RoboDK station: Prep Stacji Filip.rdk

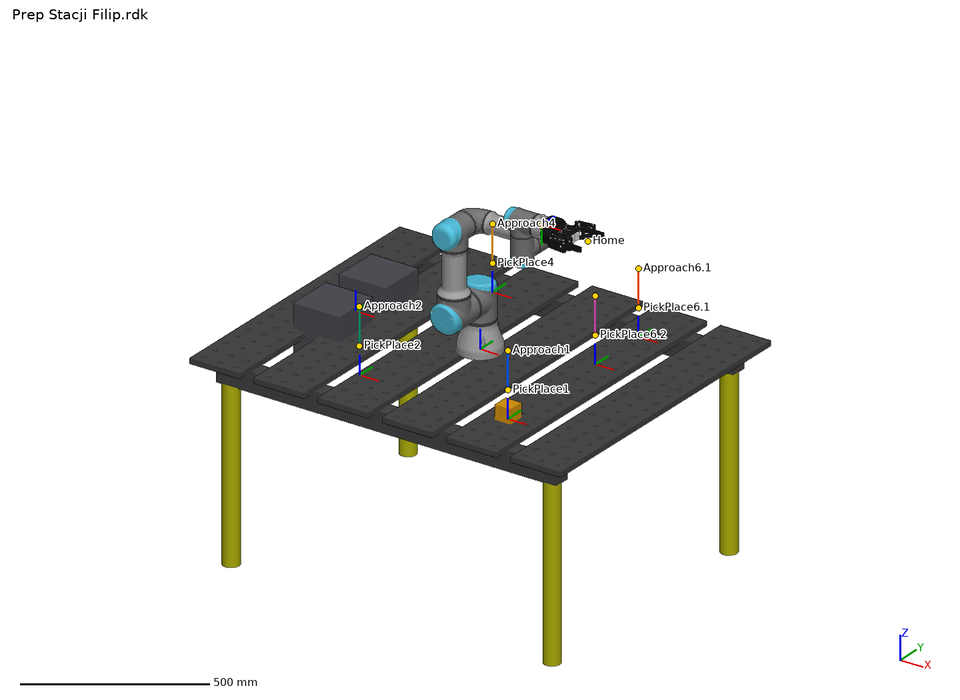
[picture v0: the station drawn from its stored meshes, robots at their saved joint values, targets as dots, program paths as lines]
Station Prep Stacji Filip. Poses are relative to the parent item; angles as X-Y-Z fixed-axis rotations.
  - frame UR3 Base at (0, 0, 0) mm
    - robot UR3: 6 axes, payload 3 kg, reach 500 mm, repeatability 0.1 mm, weight 11 kg
        modified DH rows (alpha deg, a mm, theta deg, d mm): 0, 0, 0, 151.9; 90, 0, 180, 0; 0, 243.65, 0, 0; 0, 213, 0, 110.4; -90, 0, 0, 83.4; 90, 0, 180, 82.4
        joint limits [-360, -360, -360, -360, -360, -360] to [360, 360, 360, 360, 360, 360]; home [0, -90, -90, 0, 90, 0]; saved at [0, -90, -90, 0, 90, 0]
      - tool Gripper, TCP at (0, 0, 130) mm, size 147.4 x 146.8 x 75 mm
    - object Table at (0, 0, 0) mm, size 1193.8 x 965.2 x 609.6 mm, geometry from welding_table.sld
    - target Home (Cartesian target) at (425.4, -110.4, 478.95) mm, rotated rx -90 ry 0 rz -90 deg; joints [0, -90, -90, 0, 90, 0] of UR3
    - object Vise_1 at (-400, 105, 0) mm, size 150 x 150 x 150 mm, geometry from box.sld
    - object Vise_2 at (-400, -105, 0) mm, size 150 x 150 x 150 mm, geometry from box.sld
  - frame Grab_Blank at (300, -300, 0) mm
    - target Approach1 (Cartesian target) at (0, 0, 200) mm, rotated rx 179.78 ry -0.22 rz -90 deg; joints [-29.763, -119.152, -47.872, -103.057, 89.704, -29.763] of UR3
    - target PickPlace1 (Cartesian target) at (0, 0, 85) mm, rotated rx 179.78 ry -0.22 rz -90 deg; joints [120.071, -59.59, 77.288, -107.776, -90.297, -59.929] of UR3
  - frame Blank_Buffer at (-170, -310, 0) mm
    - target Approach2 (Cartesian target) at (0, 0, 200) mm, rotated rx 179.78 ry -0.22 rz 90 deg; joints [-119.875, -118.751, -48.653, -102.3, 89.919, -119.875] of UR3
    - target PickPlace2 (Cartesian target) at (0, 0, 85) mm, rotated rx 179.78 ry -0.22 rz 90 deg; joints [-119.875, -120.162, -77.775, -71.767, 89.919, -119.875] of UR3
  - frame Workpiece_Holder at (-400, 0, 0) mm
  - frame Workpiece_Buffer at (-170, 300, 0) mm
    - target Approach4 (Cartesian target) at (0, 0, 200) mm, rotated rx 179.78 ry -0.22 rz 90 deg; joints [-209.763, -119.154, -47.869, -103.059, 89.704, -29.763] of UR3
    - target PickPlace4 (Cartesian target) at (0, 0, 85) mm, rotated rx 179.78 ry -0.22 rz 90 deg; joints [-209.763, -120.393, -77.248, -72.441, 89.704, -29.763] of UR3
  - frame Inspection_Point at (-47.33, 351.68, 211.92) mm, rotated rx -90 ry 0 rz 0 deg
    - target Inspekcja (Cartesian target) at (4.05, 0, -6.89) mm, rotated rx 0 ry 1.16 rz 0 deg; joints [161.436, -62.355, -137.519, -160.126, -17.407, 180] of UR3
    - target Inspekcja2 (Cartesian target) at (4.12, -0.12, -6.97) mm, rotated rx -0.02 ry -1.17 rz -180 deg; joints [161.482, -62.272, -137.542, -160.119, -17.348, -0.064] of UR3
    - target Inspekcja3 (Cartesian target) at (4.12, -0.12, -6.97) mm, rotated rx 0.02 ry 1.17 rz 0.01 deg; joints [161.482, -62.272, -137.542, -160.119, -17.348, 179.946] of UR3
  - frame Reject_Workpiece at (300, 300, 0) mm
    - target Approach6.1 (Cartesian target) at (0, 0, 200) mm, rotated rx 179.78 ry -0.22 rz -90 deg; joints [60.042, -119.541, -47.172, -103.583, 90.08, 60.041] of UR3
    - target PickPlace6.1 (Cartesian target) at (0, 0, 85) mm, rotated rx 179.78 ry -0.22 rz -90 deg; joints [60.042, -120.641, -76.761, -72.895, 90.08, 60.041] of UR3
  - frame Approve_Workpiece at (300, 100, 0) mm
    - target Approach6.2 (Cartesian target) at (0, 0, 200) mm, rotated rx 179.78 ry -0.22 rz -90 deg; joints [38.892, -90.405, -84.937, -94.964, 89.967, 38.892] of UR3
    - target PickPlace6.2 (Cartesian target) at (0, 0, 85) mm, rotated rx 179.78 ry -0.22 rz -90 deg; joints [38.892, -95.685, -111.257, -63.363, 89.967, 38.892] of UR3
  - program ResetStation (1 instructions, listed below)
  - program Pick1 (6 instructions, listed below)
  - program Pick2 (6 instructions, listed below)
  - program Place2 (6 instructions, listed below)
  - program Pick4 (6 instructions, listed below)
  - program Place4 (6 instructions, listed below)
  - program Inspekcja (5 instructions, listed below)
  - program Pick6.1 (6 instructions, listed below)
  - program Place6.1 (6 instructions, listed below)
  - program Pick6.2 (6 instructions, listed below)
  - program Place6.2 (6 instructions, listed below)
  - program main (8 instructions, listed below)
  - object Workpiece_50mm at (300, -300, 20) mm, size 50 x 50 x 50 mm, geometry from box.sld
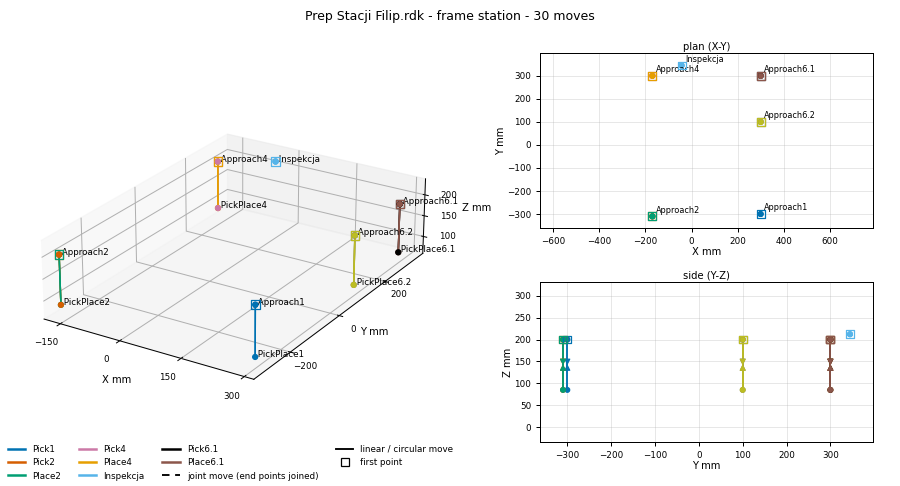
[picture p0: tool path of Prep Stacji Filip.rdk in frame station, 30 of 30 moves have a stored position in this frame; points joined in program order, loops and branches not executed]

--- program ResetStation (robot UR3) ---
  Replace Workpiece_50mm

--- program Pick1 (robot UR3) ---
  Set Ref.: Pos1 -> Grab_Blank
  Set Tool: Gripper
  MoveJ (Approach1)
  MoveL (PickPlace1)
  Attach to Gripper
  MoveL (Approach1)

--- program Pick2 (robot UR3) ---
  Set Ref.: Pos2 -> Blank_Buffer
  Set Tool: Gripper
  MoveJ (Approach2)
  MoveL (PickPlace2)
  Attach to Gripper
  MoveL (Approach2)

--- program Place2 (robot UR3) ---
  Set Ref.: Pos2 -> Blank_Buffer
  Set Tool: Gripper
  MoveJ (Approach2)
  MoveL (PickPlace2)
  Detach from Gripper
  MoveL (Approach2)

--- program Pick4 (robot UR3) ---
  Set Ref.: Pos4 -> Workpiece_Buffer
  Set Tool: Gripper
  MoveJ (Approach4)
  MoveL (PickPlace4)
  Attach to Gripper
  MoveL (Approach4)

--- program Place4 (robot UR3) ---
  Set Ref.: Pos4 -> Workpiece_Buffer
  Set Tool: Gripper
  MoveJ (Approach4)
  MoveL (PickPlace4)
  Detach from Gripper
  MoveL (Approach4)

--- program Inspekcja (robot UR3) ---
  Set Ref.: Frame 6 -> Inspection_Point
  Set Tool: Gripper
  MoveJ (Inspekcja)
  MoveJ (Inspekcja2)
  MoveJ (Inspekcja3)

--- program Pick6.1 (robot UR3) ---
  Set Ref.: Pos6.1 -> Reject_Workpiece
  Set Tool: Gripper
  MoveJ (Approach6.1)
  MoveL (PickPlace6.1)
  Attach to Gripper
  MoveL (Approach6.1)

--- program Place6.1 (robot UR3) ---
  Set Ref.: Pos6.1 -> Reject_Workpiece
  Set Tool: Gripper
  MoveJ (Approach6.1)
  MoveL (PickPlace6.1)
  Detach from Gripper
  MoveL (Approach6.1)

--- program Pick6.2 (robot UR3) ---
  Set Ref.: Pos6.2 -> Approve_Workpiece
  Set Tool: Gripper
  MoveJ (Approach6.2)
  MoveL (PickPlace6.2)
  Attach to Gripper
  MoveL (Approach6.2)

--- program Place6.2 (robot UR3) ---
  Set Ref.: Pos6.2 -> Approve_Workpiece
  Set Tool: Gripper
  MoveJ (Approach6.2)
  MoveL (PickPlace6.2)
  Detach from Gripper
  MoveL (Approach6.2)

--- program main (robot UR3) ---
  Call ResetStation
  Call Pick1
  Call Place2
  Call Pick2
  Call Place4
  Call Pick4
  Call Inspekcja
  Call Place6.1
